FUNCTION_BLOCK SoEResetTask IMPLEMENTS I_Task, I_Cyclic, I_Object, I_Abortable, I_Abortable, I_Resettable
VAR
	fbSoEReset : FB_SoEReset;
	mcReset : Tc2_MC2.MC_Reset;
	_Axis : REFERENCE TO Tc2_MC2.AXIS_REF;
	State: INT;
END_VAR

METHOD Abort : HRESULT
fbSoEReset.Execute := FALSE;
mcReset.Execute := FALSE;
State := 0;
END_METHOD

PROPERTY AxisRef : reference to Axis_Ref
GET // PUBLIC
AxisRef REF= _Axis;
END_GET
SET
_Axis REF= AxisRef;
END_SET
END_PROPERTY

PROPERTY Busy : BOOL
GET
Busy := fbSoEReset.Busy;
END_GET
END_PROPERTY

METHOD Cycle : HRESULT
IF NOT __ISVALIDREF(_Axis) THEN
	Cycle := -1;
	RETURN;
END_IF

CASE State OF
	10:
		fbSoEReset.Execute := TRUE;
		State := State + 10;
	20:
		IF NOT fbSoEReset.Busy THEN
			State := State + 10;
		END_IF
	30:
		mcReset.Execute := TRUE;
		State := State + 10;
	40:
		IF mcReset.Done THEN
			State := 0;
		END_IF
END_CASE

mcReset(Axis := _Axis);
mcReset.Execute := FALSE;
fbSoEReset(Axis := _Axis);
fbSoEReset.Execute := FALSE;
END_METHOD

PROPERTY Done : BOOL
GET
Done := NOT fbSoEReset.Busy;
END_GET
END_PROPERTY

PROPERTY Error : BOOL
GET
Error := fbSoEReset.Error;
END_GET
END_PROPERTY

METHOD RegisterWithParent
VAR_INPUT
	Parent	: I_HostObjects;
END_VAR
Parent.RegisterAbortable(THIS^);
Parent.RegisterCyclic(THIS^);
Parent.RegisterTask(THIS^);
Parent.RegisterResettable(THIS^);
END_METHOD

METHOD Reset : HRESULT
IF State <> 0 THEN
	Reset := -1;
	RETURN;
END_IF
State := 10;
END_METHOD

END_FUNCTION_BLOCK

(* stored: Version 1.1.0.1
   POU SoEResetTask: Id {18ee4c2b-0397-43b0-96c9-a74db5cdf638}, SpecialFunc None
   Method Abort: Id {d1b8bf4e-72b7-4caf-8c7e-6b13934f1684}
   Property AxisRef: Id {49d101db-d63e-4e1d-b960-d690830beeca}
   Get Get: Id {0de21b7a-2d14-4e71-a48c-7da84576c729}
   Set Set: Id {860fc9c4-6a89-42c6-a58a-26d3a5aa9a24}
   Property Busy: Id {10e3eb85-5b6d-4a9a-b398-e0ead7417fd3}
   Get Get: Id {0e4cba5a-f213-4c9c-a248-765dda70ddb4}
   Method Cycle: Id {3e415f12-eb0c-4594-a316-546282543fe0}
   Property Done: Id {7e17c524-4818-46ca-b7d3-c5b14f76a4ed}
   Get Get: Id {ba1507b4-0009-477a-916a-ab4a0da6c299}
   Property Error: Id {20cf0a5d-4703-475e-88cf-b97e5271c03d}
   Get Get: Id {d4e97ff5-17a6-487e-b1b3-7d5c749fcc82}
   Method RegisterWithParent: Id {1471b488-29bb-4efa-990d-7576394ede6e}
   Method Reset: Id {e58546ac-e936-4b87-896e-1c1cb4cb0c40} *)
